# EPICS substitutions: apps/mmfeuApp/Db/mmfeucrate.substitutions
#
file "db/mmfeucrate.db" {
        pattern { P, C, PORT}
                {"B_DET_MVT_FEU", "1", "L1"  }
#                {"B_DET_MVT_FEU", "2", "L1"  }
#               {"B_DET_MVT_FEU", "3", "L1"  }
#               {"B_DET_MVT_FEU", "4", "L1"  }
#               {"B_DET_MVT_FEU", "5", "L1"  }
#               {"B_DET_MVT_FEU", "6", "L1"  }
}
